TYPE ST_EtherCATMaster :
STRUCT
	nDeviceId	: WORD;
	sNetId 		: T_AmsNetID;
	nCfgSlaves	: UINT;
	aStSlaveInfo : ARRAY[0..15] OF ST_EcSlaveConfigData;
END_STRUCT
END_TYPE

(* stored: Version 1.1.0.1, ProductVersion 3.1.4022.10
   DUT ST_EtherCATMaster: Id {2c6ed391-bd58-4132-9e4c-71fbc1fbfda5} *)
